FUNCTION_BLOCK CurrOwnerDecode (* Basic Function Block Type *)
  (* Standard: 61499-2 *)
  (* Version 0.0, 6/3/2026, Schneider Electric, Template *)
  PACKAGE SE.Nereda;
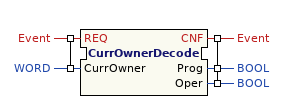
  EVENT_INPUT
    REQ WITH CurrOwner; (* Normal Execution Request *)
  END_EVENT
  EVENT_OUTPUT
    CNF WITH Prog, Oper; (* Execution Confirmation *)
  END_EVENT
  VAR_INPUT
    CurrOwner : WORD;
  END_VAR
  VAR_OUTPUT
    Prog : BOOL;
    Oper : BOOL;
  END_VAR
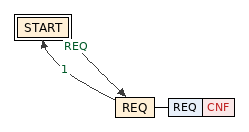
  EC_STATES
    START; (* Initial State *)
    REQ : REQ -> CNF; (* Normal execution *)
  END_STATES
  EC_TRANSITIONS
    START TO REQ := REQ;
    REQ TO START := 1;
  END_TRANSITIONS
  ALGORITHM REQ IN ST: (* Normally executed algorithm *)
;
IF CurrOwner = 16#8 OR CurrOwner = 16#4 THEN
	Prog := TRUE;
	Oper := FALSE;
ELSIF CurrOwner = 16#10 OR CurrOwner = 16#40 THEN
	Prog := FALSE;
	Oper := TRUE;
END_IF;
  END_ALGORITHM
END_FUNCTION_BLOCK
